// TIA Portal V20 export
TYPE "LER_typePartTrackingControlNode"
// stored: Access Published
   STRUCT
      command { S7_SetPoint := 'True'} : "LER_typePartTrackingCommand";
      partData { S7_SetPoint := 'True'} : "LER_typePartData";
      partStatus { S7_SetPoint := 'True'} : "LER_typePartStatus";
   END_STRUCT;
END_TYPE
